TYPE "MEStoPLC_SubCheckIn"
VERSION : 0.1
   STRUCT
      "M-SubPartDone" : Bool;
      "M-SubPartOK" : Bool;
      "M-SubPartNG" : Bool;
      "M-SubPartErrorCode" : Int;
      "M-SubPartErrorMsg" : String[98];
      Reserve : Array[1..196] of Byte;
   END_STRUCT;

END_TYPE

